TYPE st_IO_Outputs :
STRUCT
    hydroPump : ST_Pump_Output;
    robot : ST_Robot_Output;
END_STRUCT
END_TYPE

(* stored: Version 1.1.0.1, ProductVersion 3.1.4024.9
   DUT st_IO_Outputs: Id {20d84fad-c6da-49fc-a30b-ccfc3c24ee24} *)
